// TIA Portal V18 export
// export: Created 2026-01-09T11:31:52.7292056Z, ExportSetting WithDefaults, DisplayName Totally Integrated Automation Portal, DisplayVersion V18 Update 5, DisplayName TIA Portal Openness, DisplayVersion V18 Update 5, DisplayName TIA Portal Teamcenter Gateway, DisplayVersion V18, DisplayName TIA Portal Version Control Interface, DisplayVersion V18, DisplayName SINAMICS Startdrive Advanced, DisplayVersion V18 SP2 Update 1, DisplayName SINAMICS Startdrive G110M, G120, G120C, G120D, G120P, G115D, DisplayVersion V18 SP2 Update 1, DisplayName SINAMICS Startdrive G130, G150, S120, S150, SINAMICS MV, S210, G220, S200, DisplayVersion V18 SP2 Update 1, DisplayName STEP 7 Professional, DisplayVersion V18 Update 5, DisplayName STEP 7 Safety, DisplayVersion V18, DisplayName WinCC Professional, DisplayVersion V18 Update 5
TagTable "Bar"
  TimeMin : Int  (1 s)
  TimeMax : Int  (1 s)
  CountMaxD : DInt  (1 s)
  CountMinD : DInt  (1 s)
  TimeTMax : DInt  (1 s)
  TimeTMin : DInt  (1 s)
  TimeMMax : Int  (1 s)
  TimeMMin : Int  (1 s)
